# EPICS autosave request: CameraApp/Db/camera.req
file "ADBase_settings.req",       P=$(P),     R=$(R)
file "aravisCamera_settings.req", P=$(P),     R=$(R)
file "NDStdArrays_settings.req",  P=$(P),     R=image1:
